{attribute 'qualified_only'}
{attribute 'strict'}
{attribute 'to_string'}
TYPE E_Level :
(
	enum_member := 0
);
END_TYPE

(* stored: Version 1.1.0.1
   DUT E_Level: Id {64e47300-2181-0959-1f97-e8d7a09e0815} *)
